TYPE ST_TriggerBox :
STRUCT
  // MB Triggerbox Function
  // - output to CAM at given AxisPosition
  // - input feedback from FlashController trigger timestamp
  // - input feedback of AxisPosition at timestamp (FlashPosition)
  ToPlc   : ST_TriggerSet;
  FromPlc : ST_TriggerGet;  
END_STRUCT
END_TYPE

(* stored: Version 1.1.0.1, ProductVersion 3.1.4024.12
   DUT ST_TriggerBox: Id {7bebcc89-848c-4317-a4db-001979b08fb4} *)
